FUNCTION_BLOCK FB_OCHSNER_Web2Com1_Helper
VAR_INPUT
	bSend				: BOOL;
END_VAR

VAR_IN_OUT
	fbClient			: FB_IotHttpClient;
END_VAR

VAR_OUTPUT
	bBusy				: BOOL;
	bError				: BOOL;
	byHP1StateHeatProd		: BYTE;
	lrHP1TWVtemp			: LREAL;
	lrHP1TWRtemp			: LREAL;
	lrHP1TQAtemp			: LREAL;
	lrHP1TQEtemp			: LREAL;
	lrHP1ThEnergykWh		: LREAL;
	lrHP1ThEnergyMWh		: LREAL;
	byHC1StateHC			: BYTE;
	lrHC1OutTemp			: LREAL;
	lrHC1OutTempAvg			: LREAL;
	lrHC1SPRoomTemp			: LREAL;
	lrHC1PreFlowTemp		: LREAL;
	lrHC1SPFlowTemp			: LREAL;
	byHP2StateHeatProd		: BYTE;
	lrHP2TWVtemp			: LREAL;
	lrHP2TWRtemp			: LREAL;
	lrHP2TQAtemp			: LREAL;
	lrHP2TQEtemp			: LREAL;
	lrHP2ThEnergykWh		: LREAL;
	lrHP2ThEnergyMWh		: LREAL;
END_VAR

VAR
	fbRequest1			: FB_IotHttpRequest;
	fbRequest2			: FB_IotHttpRequest;
	fbRequest3			: FB_IotHttpRequest;

	fbJson				: FB_JsonDomParser;
	nState				: UDINT;
	RisingEdge			: R_TRIG;
	timTimeout			: TON;
	tTimeOut			: TIME := T#90S;
	bGetContentResult	: BOOL;
	sContent1			: STRING(511);
	sContent2			: STRING(511);
	sContent3			: STRING(511);
	
	bGetJsonResult		: BOOL;
	jsonDoc				: SJsonValue;
	jsonVal				: SJsonValue;
	
	nReqCount			: UDINT;	
	nResCount			: UDINT;
	nValidResCount		: UDINT;
	nErrCount			: UDINT;
END_VAR

//Timer for Timeout
timTimeout(IN:= nState = 1 AND bBusy, PT:= tTimeOut, Q=> , ET=> );
	IF timTimeout.Q THEN 
		nState := 0;
		bBusy := FALSE;
	END_IF

RisingEdge(CLK:= bSend );
CASE nState OF
0:	
	IF RisingEdge.Q THEN 
		IF 
			fbRequest1.SendRequest(sUri:='/web2com_1HP1.php', fbClient:=fbClient, eRequestType:=ETcIotHttpRequestType.HTTP_Get, 0, 0, 0) AND
			fbRequest2.SendRequest(sUri:='/web2com_1HC1.php', fbClient:=fbClient, eRequestType:=ETcIotHttpRequestType.HTTP_Get, 0, 0, 0) AND 
			fbRequest3.SendRequest(sUri:='/web2com_1HP2.php', fbClient:=fbClient, eRequestType:=ETcIotHttpRequestType.HTTP_Get, 0, 0, 0) THEN				
			nState:= 1;
			nReqCount:= nReqCount+1;
			bBusy:= TRUE;
			bError:= FALSE;
		END_IF					
	END_IF
1:
	IF NOT fbRequest1.bBusy AND NOT fbRequest2.bBusy AND NOT fbRequest3.bBusy THEN
		bError:= TRUE;
		IF NOT fbRequest1.bError THEN				 
			bGetContentResult:= fbRequest1.GetContent(pContent:= ADR(sContent1), nContentSize:= SIZEOF(sContent1), bSetNullTermination:= TRUE);
			IF fbRequest1.nStatusCode >= 200 AND fbRequest1.nStatusCode < 300 THEN
				bGetJsonResult:= FALSE;
				jsonDoc:= fbRequest1.GetJsonDomContent(fbJson);
				IF jsonDoc <> 0 THEN
					bGetJsonResult:= TRUE;
					IF fbJson.HasMember(jsonDoc, '1211250')  THEN
						jsonVal:= fbJson.FindMember(jsonDoc, '1211250');
						nValidResCount:= nValidResCount+1;
						IF fbJson.IsNumber(jsonVal) THEN							
							byHP1StateHeatProd := DINT_TO_BYTE(fbJson.GetInt(jsonVal));									
						END_IF
						
						jsonVal:= fbJson.FindMember(jsonDoc, '1211251');
						nValidResCount:= nValidResCount+1;
						IF fbJson.IsDouble(jsonVal) THEN							
							lrHP1TWVtemp := fbJson.GetDouble(jsonVal);									
						END_IF
						
						jsonVal:= fbJson.FindMember(jsonDoc, '1211253');
						nValidResCount:= nValidResCount+1;
						IF fbJson.IsDouble(jsonVal) THEN							
							lrHP1TWRtemp := fbJson.GetDouble(jsonVal);									
						END_IF
						
						jsonVal:= fbJson.FindMember(jsonDoc, '1211254');
						nValidResCount:= nValidResCount+1;
						IF fbJson.IsDouble(jsonVal) THEN							
							lrHP1TQAtemp := fbJson.GetDouble(jsonVal);									
						END_IF
						
						jsonVal:= fbJson.FindMember(jsonDoc, '1211255');
						nValidResCount:= nValidResCount+1;
						IF fbJson.IsDouble(jsonVal) THEN							
							lrHP1TQEtemp := fbJson.GetDouble(jsonVal);									
						END_IF
						
						jsonVal:= fbJson.FindMember(jsonDoc, '1211258');
						nValidResCount:= nValidResCount+1;
						IF fbJson.IsNumber(jsonVal) THEN							
							lrHP1ThEnergykWh := fbJson.GetDouble(jsonVal);									
						END_IF
						
						jsonVal:= fbJson.FindMember(jsonDoc, '1211259');
						nValidResCount:= nValidResCount+1;
						IF fbJson.IsNumber(jsonVal) THEN							
							lrHP1ThEnergyMWh := fbJson.GetDouble(jsonVal);									
						END_IF
						
						bError:= FALSE;
						END_IF
					END_IF						
				nResCount:= nResCount+1;			
				END_IF
		END_IF
		
		IF NOT fbRequest2.bError THEN				 
			bGetContentResult:= fbRequest2.GetContent(pContent:= ADR(sContent2), nContentSize:= SIZEOF(sContent2), bSetNullTermination:= TRUE);
			IF fbRequest2.nStatusCode >= 200 AND fbRequest2.nStatusCode < 300 THEN
				bGetJsonResult:= FALSE;
				jsonDoc:= fbRequest2.GetJsonDomContent(fbJson);
				IF jsonDoc <> 0 THEN
					bGetJsonResult:= TRUE;
					IF fbJson.HasMember(jsonDoc, '1241190')  THEN
						jsonVal:= fbJson.FindMember(jsonDoc, '1241190');
						nValidResCount:= nValidResCount+1;
						IF fbJson.IsNumber(jsonVal) THEN							
							byHC1StateHC := DINT_TO_BYTE(fbJson.GetInt(jsonVal));									
						END_IF
						
						jsonVal:= fbJson.FindMember(jsonDoc, '1241191');
						nValidResCount:= nValidResCount+1;
						IF fbJson.IsDouble(jsonVal) THEN							
							lrHC1OutTemp := fbJson.GetDouble(jsonVal);									
						END_IF
						
						jsonVal:= fbJson.FindMember(jsonDoc, '1241192');
						nValidResCount:= nValidResCount+1;
						IF fbJson.IsDouble(jsonVal) THEN							
							lrHC1OutTempAvg := fbJson.GetDouble(jsonVal);									
						END_IF
						
						jsonVal:= fbJson.FindMember(jsonDoc, '1241193');
						nValidResCount:= nValidResCount+1;
						IF fbJson.IsDouble(jsonVal) THEN							
							lrHC1SPRoomTemp := fbJson.GetDouble(jsonVal);									
						END_IF
						
						jsonVal:= fbJson.FindMember(jsonDoc, '1241194');
						nValidResCount:= nValidResCount+1;
						IF fbJson.IsDouble(jsonVal) THEN							
							lrHC1PreFlowTemp := fbJson.GetDouble(jsonVal);									
						END_IF
						
						jsonVal:= fbJson.FindMember(jsonDoc, '1241195');
						nValidResCount:= nValidResCount+1;
						IF fbJson.IsDouble(jsonVal) THEN							
							lrHC1SPFlowTemp := fbJson.GetDouble(jsonVal);									
						END_IF
						
						bError:= FALSE;
						END_IF
					END_IF						
				nResCount:= nResCount+1;			
				END_IF
		END_IF
		
		IF NOT fbRequest3.bError THEN				 
			bGetContentResult:= fbRequest3.GetContent(pContent:= ADR(sContent3), nContentSize:= SIZEOF(sContent3), bSetNullTermination:= TRUE);
			IF fbRequest3.nStatusCode >= 200 AND fbRequest3.nStatusCode < 300 THEN
				bGetJsonResult:= FALSE;
				jsonDoc:= fbRequest3.GetJsonDomContent(fbJson);
				IF jsonDoc <> 0 THEN
					bGetJsonResult:= TRUE;
					IF fbJson.HasMember(jsonDoc, '1311250')  THEN
						jsonVal:= fbJson.FindMember(jsonDoc, '1311250');
						nValidResCount:= nValidResCount+1;
						IF fbJson.IsNumber(jsonVal) THEN							
							byHP2StateHeatProd := DINT_TO_BYTE(fbJson.GetInt(jsonVal));									
						END_IF
						
						jsonVal:= fbJson.FindMember(jsonDoc, '1311251');
						nValidResCount:= nValidResCount+1;
						IF fbJson.IsDouble(jsonVal) THEN							
							lrHP2TWVtemp := fbJson.GetDouble(jsonVal);									
						END_IF
						
						jsonVal:= fbJson.FindMember(jsonDoc, '1311253');
						nValidResCount:= nValidResCount+1;
						IF fbJson.IsDouble(jsonVal) THEN							
							lrHP2TWRtemp := fbJson.GetDouble(jsonVal);									
						END_IF
						
						jsonVal:= fbJson.FindMember(jsonDoc, '1311254');
						nValidResCount:= nValidResCount+1;
						IF fbJson.IsDouble(jsonVal) THEN							
							lrHP2TQAtemp := fbJson.GetDouble(jsonVal);									
						END_IF
						
						jsonVal:= fbJson.FindMember(jsonDoc, '1311255');
						nValidResCount:= nValidResCount+1;
						IF fbJson.IsDouble(jsonVal) THEN							
							lrHP2TQEtemp := fbJson.GetDouble(jsonVal);									
						END_IF
						
						jsonVal:= fbJson.FindMember(jsonDoc, '1311258');
						nValidResCount:= nValidResCount+1;
						IF fbJson.IsNumber(jsonVal) THEN							
							lrHP2ThEnergykWh := fbJson.GetDouble(jsonVal);									
						END_IF
						
						jsonVal:= fbJson.FindMember(jsonDoc, '1311259');
						nValidResCount:= nValidResCount+1;
						IF fbJson.IsNumber(jsonVal) THEN							
							lrHP2ThEnergyMWh := fbJson.GetDouble(jsonVal);									
						END_IF
						
						bError:= FALSE;
						END_IF
					END_IF						
				nResCount:= nResCount+1;			
				END_IF
		END_IF
		
		nState:= 0;
		bBusy:= FALSE;
		IF bError THEN
			nErrCount:= nErrCount+1;
		END_IF
	END_IF  	
END_CASE

END_FUNCTION_BLOCK

(* stored: Version 1.1.0.1, ProductVersion 3.1.4024.11
   POU FB_OCHSNER_Web2Com1_Helper: Id {d52dbd3e-7205-46d1-ad6e-a7882bd17748}, SpecialFunc None *)
